TYPE
    ST_SetupFanucRobot :
    STRUCT
        RobotVelocity : LREAL :=20 ;
		ZoneCCD : ST_FanucRobotCCDSetting;
    END_STRUCT
END_TYPE

(* stored: Version 1.1.0.1, ProductVersion 3.1.4024.13
   DUT ST_SetupFanucRobot: Id {97c13032-e5a3-42af-870a-87f988859e63} *)
